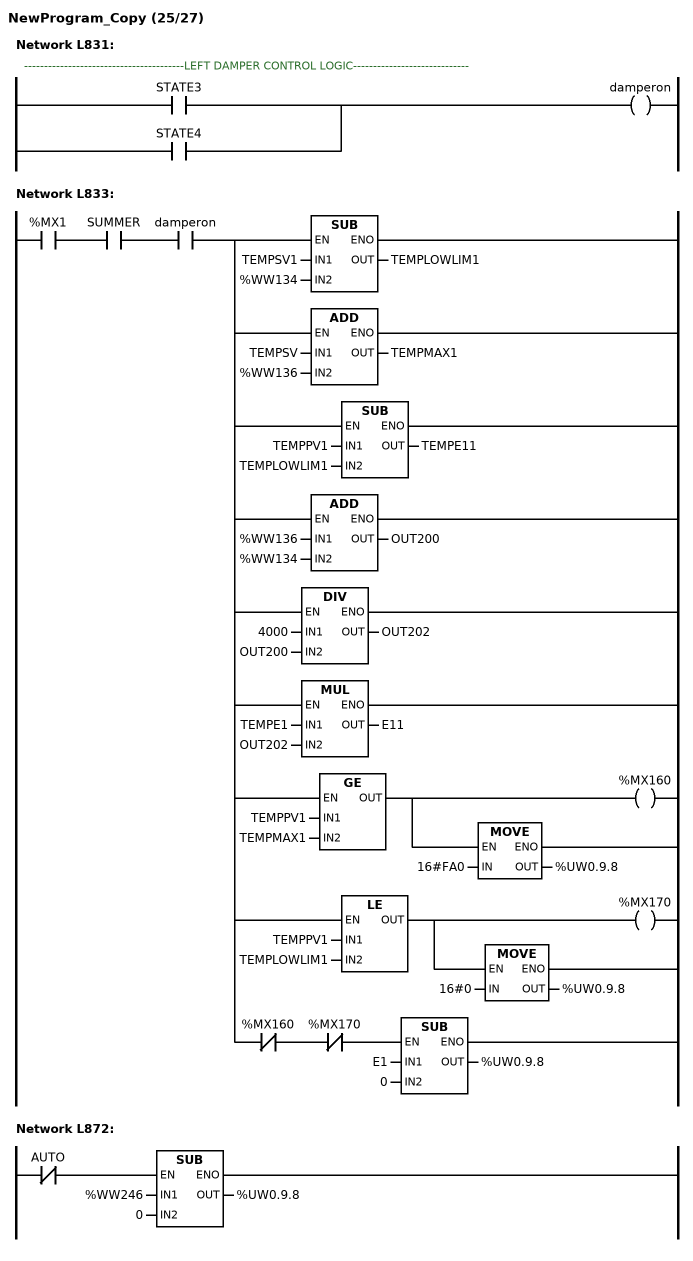
(* [picture p24: NewProgram_Copy rungs L831-L872] *)
(* ----------------------------------------LEFT DAMPER CONTROL LOGIC----------------------------- *)
(* Rung L831 *)
damperon := STATE3 OR STATE4;
(* Rung L833 *)
IF %MX1 AND SUMMER AND damperon THEN
    TEMPLOWLIM1 := TEMPSV1 - %WW134;
    TEMPMAX1 := TEMPSV + %WW136;
    TEMPE11 := TEMPPV1 - TEMPLOWLIM1;
    OUT200 := %WW136 + %WW134;
    OUT202 := 4000 / OUT200;
    E11 := TEMPE1 * OUT202;
    _t35 := TEMPPV1 >= TEMPMAX1;
END_IF;
%MX160 := _t35;
IF _t35 THEN %UW0.9.8 := 16#FA0; END_IF;
IF %MX1 AND SUMMER AND damperon THEN _t36 := TEMPPV1 <= TEMPLOWLIM1; END_IF;
%MX170 := _t36;
IF _t36 THEN %UW0.9.8 := 16#0; END_IF;
IF %MX1 AND SUMMER AND damperon AND NOT %MX160 AND NOT %MX170 THEN %UW0.9.8 := E1 - 0; END_IF;
(* Rung L872 *)
IF NOT AUTO THEN %UW0.9.8 := %WW246 - 0; END_IF;

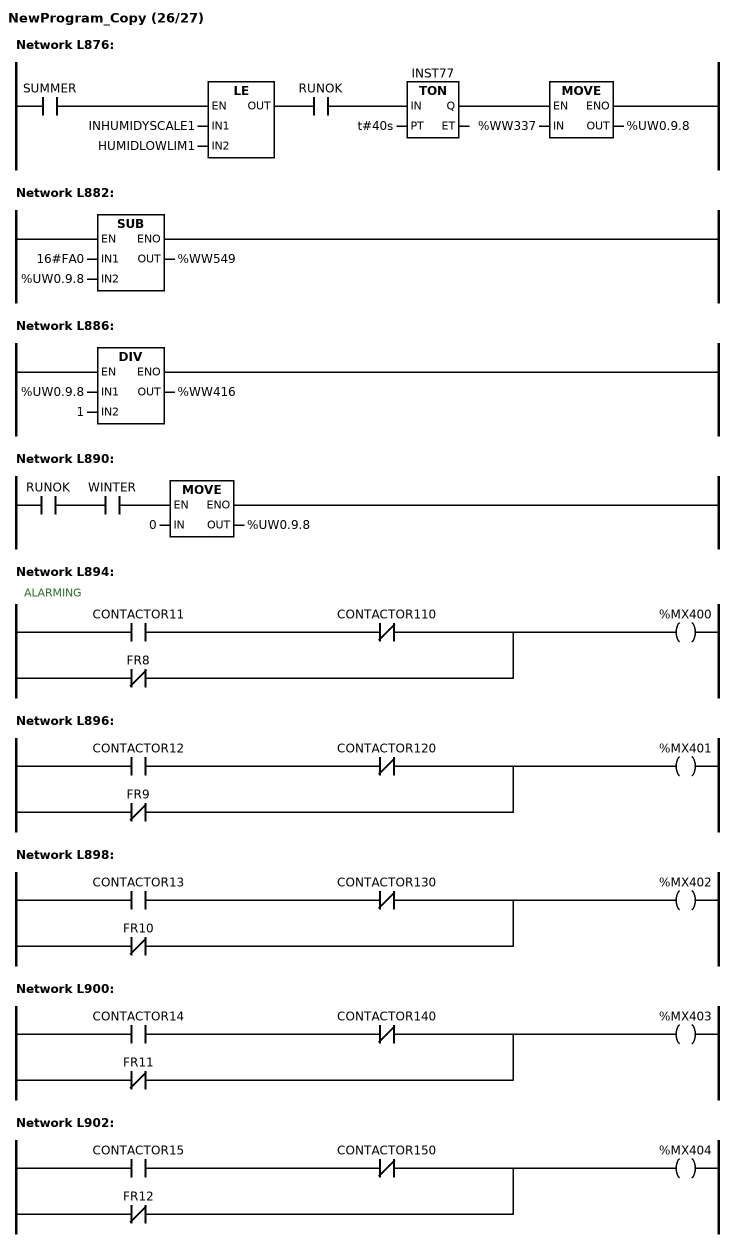
(* Rung L876 *)
IF SUMMER THEN _t37 := INHUMIDYSCALE1 <= HUMIDLOWLIM1; END_IF;
INST77(IN := _t37 AND RUNOK, PT := t#40s);
IF INST77.Q THEN %UW0.9.8 := %WW337; END_IF;
(* Rung L882 *)
%WW549 := 16#FA0 - %UW0.9.8;
(* Rung L886 *)
%WW416 := %UW0.9.8 / 1;
(* Rung L890 *)
IF RUNOK AND WINTER THEN %UW0.9.8 := 0; END_IF;
(* ALARMING *)
(* Rung L894 *)
%MX400 := (CONTACTOR11 AND NOT CONTACTOR110) OR NOT FR8;
(* Rung L896 *)
%MX401 := (CONTACTOR12 AND NOT CONTACTOR120) OR NOT FR9;
(* Rung L898 *)
%MX402 := (CONTACTOR13 AND NOT CONTACTOR130) OR NOT FR10;
(* Rung L900 *)
%MX403 := (CONTACTOR14 AND NOT CONTACTOR140) OR NOT FR11;
(* Rung L902 *)
%MX404 := (CONTACTOR15 AND NOT CONTACTOR150) OR NOT FR12;

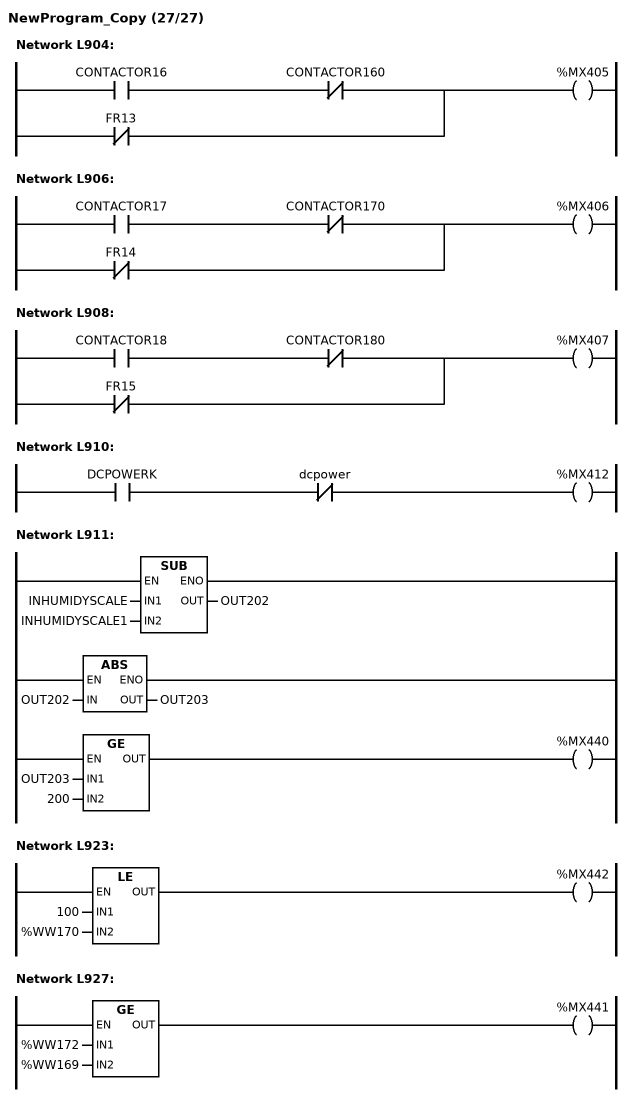
(* Rung L904 *)
%MX405 := (CONTACTOR16 AND NOT CONTACTOR160) OR NOT FR13;
(* Rung L906 *)
%MX406 := (CONTACTOR17 AND NOT CONTACTOR170) OR NOT FR14;
(* Rung L908 *)
%MX407 := (CONTACTOR18 AND NOT CONTACTOR180) OR NOT FR15;
(* Rung L910 *)
%MX412 := DCPOWERK AND NOT dcpower;
(* Rung L911 *)
OUT202 := INHUMIDYSCALE - INHUMIDYSCALE1;
OUT203 := ABS(OUT202);
%MX440 := OUT203 >= 200;
(* Rung L923 *)
%MX442 := 100 <= %WW170;
(* Rung L927 *)
%MX441 := %WW172 >= %WW169;
END_PROGRAM